TYPE sMoverPosition :
STRUCT
	x : LREAL;
	y : LREAL;
	z : LREAL;
	a : LREAL;
	b : LREAL;
	c : LREAL;
END_STRUCT
END_TYPE

(* stored: Version 1.1.0.1
   DUT sMoverPosition: Id {7524b54d-9c54-45a0-bc79-4a124e78eea7} *)
